{attribute 'TcLinkTo'}
VAR_GLOBAL
	Stepper1 : AXIS_REF;
	Stepper2 : AXIS_REF;
	Stepper3 : AXIS_REF;
	Stepper4 : AXIS_REF;
	
	Stepper_Rail1 : ST_LinearTable := (
		object := Stepper1,
		bProx := ADR(Axis1_Prox)
		);
	
	Stepper_Rail2 : ST_LinearTable := (
		object := Stepper2,
		bProx := ADR(Axis2_Prox)
		);
	
	Stepper_Rail3 : ST_LinearTable := (
		object := Stepper3,
		bProx := ADR(Axis3_Prox)
		);
	
	Stepper_Rail4 : ST_LinearTable := (
		object := Stepper4,
		bProx := ADR(Axis4_Prox)
		);
	
	Axis1 : FB_StepperMotor(init_axis := ADR(Stepper_Rail1.object));
    Axis2 : FB_StepperMotor(init_axis := ADR(Stepper_Rail2.object));
    Axis3 : FB_StepperMotor(init_axis := ADR(Stepper_Rail3.object));
    Axis4 : FB_StepperMotor(init_axis := ADR(Stepper_Rail4.object));
	Cha1 : ST_LinearActuator := (
		sName := 'Chariot1',
		bProxIn := ADR(Cha1_In) ,  
		bProxOut := ADR(Cha1_Out) , 
		bFwdDO := ADR(Cha1_Forward), 
		bBckwDO := ADR(Cha1_Reverse)
		);

	Axis1Command : ST_StepperMotorCommand := (
		Homing := FALSE,
		Command := 0,
		Position := -1,
		Homed := FALSE)
	;
	Axis2Command : ST_StepperMotorCommand := (
		Homing := FALSE,
		Command := 0,
		Position := -1,
		Homed := FALSE)
	;
	Axis3Command : ST_StepperMotorCommand := (
		Homing := FALSE,
		Command := 0,
		Position := -1,
		Homed := FALSE)
	;
	Axis4Command : ST_StepperMotorCommand := (
		Homing := FALSE,
		Command := 0,
		Position := -1,
		Homed := FALSE)
	;
	
	Max_Stepper_vel : LREAL := 2000;
END_VAR

(* stored: Version 1.1.0.1, ProductVersion 3.1.4026.11
   GVL GVL_Steppers: Id {fbf55f38-8215-4244-998d-826cf1c53444} *)
